PROGRAM P_Demo_F_BA_ToDate
VAR
    argStDate                      : ST_BA_Date                    ; // stDate
    fnReturn                       : DATE; // 返回值
END_VAR

// =============================================================================
// Tc3_BA2_Common.F_BA_ToDate 演示程序
// =============================================================================
// 场景：需要把 BA 库的日期与 IEC 标准 DATE 互操作（如喂给 IEC 标准时间函数）。
//
// 价值：一行 FC 替代手写 `DATE_TO_*` 链。
//
// 验证：登录 PLC 后，按例程内变量在线写值；监视输出 / 返回值，结合 §1 功能
//       简述的预期行为对照（详见配套 .md 文档 §7 业务场景）。
//
// 验证步骤：
//   1. 右键 PLC 项目下 POUs 文件夹 → Add → Existing Item → 选本 .TcPOU 文件
//   2. 引用 Tc3_BA2_Common（References → Add library）
//   3. 编译 → 登录 → 运行；按上方『验证』指引在线写值观察
// =============================================================================

fnReturn := F_BA_ToDate(
    stDate                   := argStDate
);

END_PROGRAM

(* stored: Version 1.1.0.1, ProductVersion 3.1.4024.5
   POU P_Demo_F_BA_ToDate: Id {b5c84a09-f08b-510d-a9ea-9b00eea5da05}, SpecialFunc None *)
